FUNCTION_BLOCK FB_Hopper
VAR_INPUT
	eMode			: E_MachineMode;
	
	bLIS101			: BOOL;
	bLIS102			: BOOL;
	
	bAck			: BOOL;
END_VAR
VAR_OUTPUT
	bFeederRequest	: BOOL;
	bWarning		: BOOL;
	bRefilling		: BOOL;
	
	bLowLevelTimeout	: BOOL;
	bFillTimeout	: BOOL;
END_VAR
VAR
	fbLowLevelTimer	: TON;
	fbFIllTimer		: TON;
	
	bAutoEnabled	: BOOL;
END_VAR

								// Automatic refill is allowed only during
									// STARTUP or normal RUN operati
								
bAutoEnabled := (eMode = E_MachineMode.MODE_STARTUP) OR (eMode = E_MachineMode.MODE_RUN);

//Warning Acknowledgement

IF bAck THEN
	bWarning := FALSE;
	bLowLevelTimeout := FALSE;
    bFillTimeout := FALSE;
END_IF

//Start Auto Refill

IF bAutoEnabled
	AND NOT bWarning
	AND NOT bLIS101
	AND NOT bRefilling THEN
		bRefilling := TRUE;
END_IF;

//Stop when high level is reached

IF bLIS102 THEN
    bRefilling := FALSE;
END_IF;

// Stop refilling outside permitted machine modes
IF NOT bAutoEnabled THEN
    bRefilling := FALSE;
END_IF;

// Timer 1:
// Low-level switch must recover within 30 seconds

fbLowLevelTimer(
	IN := bRefilling AND NOT bLIS101,
	PT := GVL_Config.c_tHopperLowTimeout
);

IF fbLowLevelTimer.Q THEN
    bLowLevelTimeout := TRUE;
END_IF;

// Timer 2:
// Complete filling must finish within 180 seconds

fbFillTimer(
    IN := bRefilling,
    PT := GVL_Config.c_tHopperFillTimeout
);

IF fbFillTimer.Q THEN
    bFillTimeout := TRUE;
END_IF;

// Fault handling

IF bLowLevelTimeout OR bFillTimeout THEN

    bWarning := TRUE;
    bRefilling := FALSE;

END_IF;

// Feeder motor request

bFeederRequest :=
    bRefilling
    AND bAutoEnabled
    AND NOT bWarning;

END_FUNCTION_BLOCK

(* stored: Version 1.1.0.1, ProductVersion 3.1.4024.16
   POU FB_Hopper: Id {55f7627a-b831-41d8-b2dc-081dda8da044}, SpecialFunc None *)
